TYPE ST_SCANNER_Ctrl :    //ST_SCANNER_CameraMap
STRUCT
	bProcessNewCode		: BOOL;
	bTCPTrigger			: BOOL;
	bManualTrigger		: BOOL;
	bResetStats			: BOOL;	
	
	stOptions			: ST_SCANNER_Options;
	stCameraMap			: ST_SCANNER_CtrlMapping;
END_STRUCT
END_TYPE

(* stored: Version 1.1.0.1
   DUT ST_SCANNER_Ctrl: Id {d8b1c7c7-f13e-4669-b41a-f9eda99bb635} *)
